// TIA Portal V17 export
// export: Created 2024-08-29T18:23:45.6211091Z, ExportSetting WithDefaults, DisplayName Totally Integrated Automation Portal, DisplayVersion V17 Update 7, DisplayName TIA Portal Openness, DisplayVersion V17 Update 7, DisplayName TIA Portal Version Control Interface, DisplayVersion V17, DisplayName SINAMICS Startdrive Advanced, DisplayVersion V17 SP2, DisplayName SINAMICS Startdrive G110M, G120, G120C, G120D, G120P, G115D, DisplayVersion V17 SP2, DisplayName SINAMICS Startdrive G130, G150, S120, S150, SINAMICS MV, S210, DisplayVersion V17 SP2, DisplayName STEP 7 Professional, DisplayVersion V17 Update 7, DisplayName STEP 7 Safety, DisplayVersion V17 Update 6, DisplayName WinCC Advanced / Unified PC, DisplayVersion V17 Update 7
FUNCTION "sensorStatusArr" : Void   // FC38, LAD
{ S7_Optimized_Access := 'TRUE' }
VERSION : 0.1
// stored: AutoNumber true, IsIECCheckEnabled false, SetENOAutomatically false, UDAEnableTagReadback false
   VAR_INPUT
      manualModeActive : Bool;
      automaticModeActive : Bool;
      sensorRequested : Array[0..31] of Bool;
      sensorActive : Array[0..31] of Bool;
      sensorMask : Array[0..31] of Bool;
   END_VAR
   VAR_OUTPUT
      sensorStatus : Array[0..31] of Byte;
   END_VAR
BEGIN

REGION Network 1: Status 0
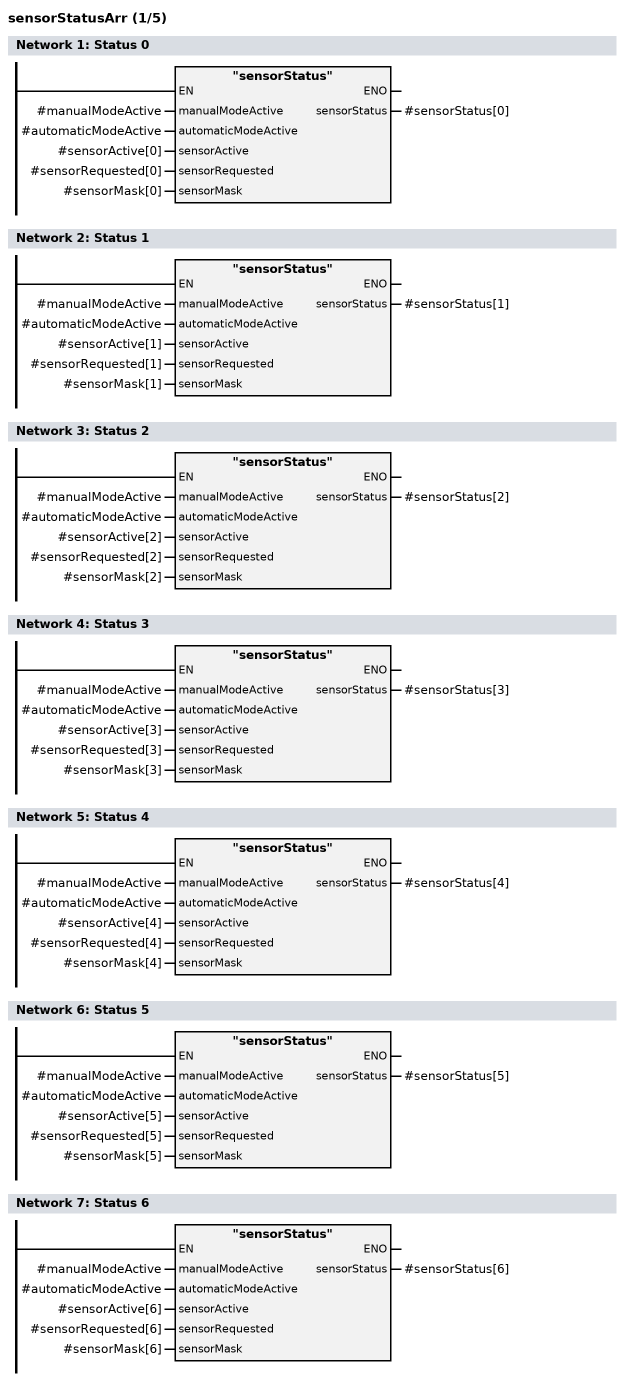
   RUNG wire#powerrail
      "sensorStatus"(manualModeActive := #manualModeActive, automaticModeActive := #automaticModeActive, sensorActive := #sensorActive[0], sensorRequested := #sensorRequested[0], sensorMask := #sensorMask[0], sensorStatus => #sensorStatus[0])
   END_RUNG
   // the same network as SCL:
   "sensorStatus"(manualModeActive := #manualModeActive,
                  automaticModeActive := #automaticModeActive,
                  sensorActive := #sensorActive[0],
                  sensorRequested := #sensorRequested[0],
                  sensorMask := #sensorMask[0],
                  sensorStatus => #sensorStatus[0]);
END_REGION

REGION Network 2: Status 1
   RUNG wire#powerrail
      "sensorStatus"(manualModeActive := #manualModeActive, automaticModeActive := #automaticModeActive, sensorActive := #sensorActive[1], sensorRequested := #sensorRequested[1], sensorMask := #sensorMask[1], sensorStatus => #sensorStatus[1])
   END_RUNG
   // the same network as SCL:
   "sensorStatus"(manualModeActive := #manualModeActive,
                  automaticModeActive := #automaticModeActive,
                  sensorActive := #sensorActive[1],
                  sensorRequested := #sensorRequested[1],
                  sensorMask := #sensorMask[1],
                  sensorStatus => #sensorStatus[1]);
END_REGION

REGION Network 3: Status 2
   RUNG wire#powerrail
      "sensorStatus"(manualModeActive := #manualModeActive, automaticModeActive := #automaticModeActive, sensorActive := #sensorActive[2], sensorRequested := #sensorRequested[2], sensorMask := #sensorMask[2], sensorStatus => #sensorStatus[2])
   END_RUNG
   // the same network as SCL:
   "sensorStatus"(manualModeActive := #manualModeActive,
                  automaticModeActive := #automaticModeActive,
                  sensorActive := #sensorActive[2],
                  sensorRequested := #sensorRequested[2],
                  sensorMask := #sensorMask[2],
                  sensorStatus => #sensorStatus[2]);
END_REGION

REGION Network 4: Status 3
   RUNG wire#powerrail
      "sensorStatus"(manualModeActive := #manualModeActive, automaticModeActive := #automaticModeActive, sensorActive := #sensorActive[3], sensorRequested := #sensorRequested[3], sensorMask := #sensorMask[3], sensorStatus => #sensorStatus[3])
   END_RUNG
   // the same network as SCL:
   "sensorStatus"(manualModeActive := #manualModeActive,
                  automaticModeActive := #automaticModeActive,
                  sensorActive := #sensorActive[3],
                  sensorRequested := #sensorRequested[3],
                  sensorMask := #sensorMask[3],
                  sensorStatus => #sensorStatus[3]);
END_REGION

REGION Network 5: Status 4
   RUNG wire#powerrail
      "sensorStatus"(manualModeActive := #manualModeActive, automaticModeActive := #automaticModeActive, sensorActive := #sensorActive[4], sensorRequested := #sensorRequested[4], sensorMask := #sensorMask[4], sensorStatus => #sensorStatus[4])
   END_RUNG
   // the same network as SCL:
   "sensorStatus"(manualModeActive := #manualModeActive,
                  automaticModeActive := #automaticModeActive,
                  sensorActive := #sensorActive[4],
                  sensorRequested := #sensorRequested[4],
                  sensorMask := #sensorMask[4],
                  sensorStatus => #sensorStatus[4]);
END_REGION

REGION Network 6: Status 5
   RUNG wire#powerrail
      "sensorStatus"(manualModeActive := #manualModeActive, automaticModeActive := #automaticModeActive, sensorActive := #sensorActive[5], sensorRequested := #sensorRequested[5], sensorMask := #sensorMask[5], sensorStatus => #sensorStatus[5])
   END_RUNG
   // the same network as SCL:
   "sensorStatus"(manualModeActive := #manualModeActive,
                  automaticModeActive := #automaticModeActive,
                  sensorActive := #sensorActive[5],
                  sensorRequested := #sensorRequested[5],
                  sensorMask := #sensorMask[5],
                  sensorStatus => #sensorStatus[5]);
END_REGION

REGION Network 7: Status 6
   RUNG wire#powerrail
      "sensorStatus"(manualModeActive := #manualModeActive, automaticModeActive := #automaticModeActive, sensorActive := #sensorActive[6], sensorRequested := #sensorRequested[6], sensorMask := #sensorMask[6], sensorStatus => #sensorStatus[6])
   END_RUNG
   // the same network as SCL:
   "sensorStatus"(manualModeActive := #manualModeActive,
                  automaticModeActive := #automaticModeActive,
                  sensorActive := #sensorActive[6],
                  sensorRequested := #sensorRequested[6],
                  sensorMask := #sensorMask[6],
                  sensorStatus => #sensorStatus[6]);
END_REGION

REGION Network 8: Status 7
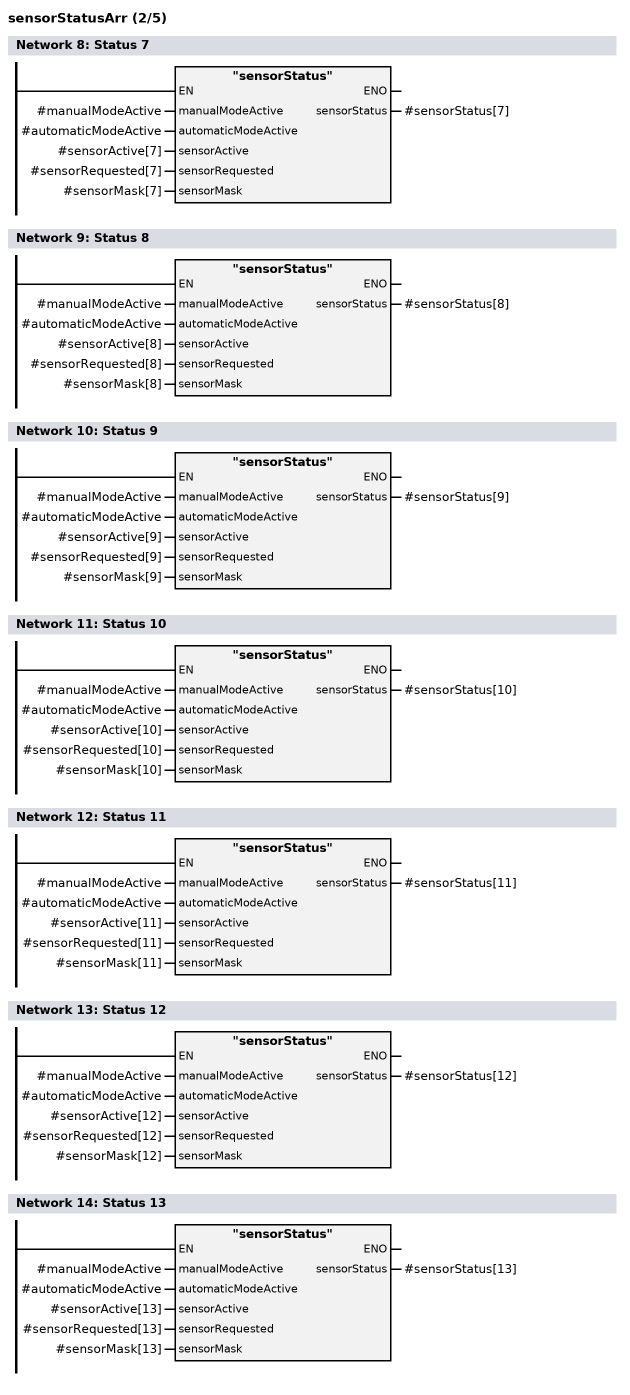
   RUNG wire#powerrail
      "sensorStatus"(manualModeActive := #manualModeActive, automaticModeActive := #automaticModeActive, sensorActive := #sensorActive[7], sensorRequested := #sensorRequested[7], sensorMask := #sensorMask[7], sensorStatus => #sensorStatus[7])
   END_RUNG
   // the same network as SCL:
   "sensorStatus"(manualModeActive := #manualModeActive,
                  automaticModeActive := #automaticModeActive,
                  sensorActive := #sensorActive[7],
                  sensorRequested := #sensorRequested[7],
                  sensorMask := #sensorMask[7],
                  sensorStatus => #sensorStatus[7]);
END_REGION

REGION Network 9: Status 8
   RUNG wire#powerrail
      "sensorStatus"(manualModeActive := #manualModeActive, automaticModeActive := #automaticModeActive, sensorActive := #sensorActive[8], sensorRequested := #sensorRequested[8], sensorMask := #sensorMask[8], sensorStatus => #sensorStatus[8])
   END_RUNG
   // the same network as SCL:
   "sensorStatus"(manualModeActive := #manualModeActive,
                  automaticModeActive := #automaticModeActive,
                  sensorActive := #sensorActive[8],
                  sensorRequested := #sensorRequested[8],
                  sensorMask := #sensorMask[8],
                  sensorStatus => #sensorStatus[8]);
END_REGION

REGION Network 10: Status 9
   RUNG wire#powerrail
      "sensorStatus"(manualModeActive := #manualModeActive, automaticModeActive := #automaticModeActive, sensorActive := #sensorActive[9], sensorRequested := #sensorRequested[9], sensorMask := #sensorMask[9], sensorStatus => #sensorStatus[9])
   END_RUNG
   // the same network as SCL:
   "sensorStatus"(manualModeActive := #manualModeActive,
                  automaticModeActive := #automaticModeActive,
                  sensorActive := #sensorActive[9],
                  sensorRequested := #sensorRequested[9],
                  sensorMask := #sensorMask[9],
                  sensorStatus => #sensorStatus[9]);
END_REGION

REGION Network 11: Status 10
   RUNG wire#powerrail
      "sensorStatus"(manualModeActive := #manualModeActive, automaticModeActive := #automaticModeActive, sensorActive := #sensorActive[10], sensorRequested := #sensorRequested[10], sensorMask := #sensorMask[10], sensorStatus => #sensorStatus[10])
   END_RUNG
   // the same network as SCL:
   "sensorStatus"(manualModeActive := #manualModeActive,
                  automaticModeActive := #automaticModeActive,
                  sensorActive := #sensorActive[10],
                  sensorRequested := #sensorRequested[10],
                  sensorMask := #sensorMask[10],
                  sensorStatus => #sensorStatus[10]);
END_REGION

REGION Network 12: Status 11
   RUNG wire#powerrail
      "sensorStatus"(manualModeActive := #manualModeActive, automaticModeActive := #automaticModeActive, sensorActive := #sensorActive[11], sensorRequested := #sensorRequested[11], sensorMask := #sensorMask[11], sensorStatus => #sensorStatus[11])
   END_RUNG
   // the same network as SCL:
   "sensorStatus"(manualModeActive := #manualModeActive,
                  automaticModeActive := #automaticModeActive,
                  sensorActive := #sensorActive[11],
                  sensorRequested := #sensorRequested[11],
                  sensorMask := #sensorMask[11],
                  sensorStatus => #sensorStatus[11]);
END_REGION

REGION Network 13: Status 12
   RUNG wire#powerrail
      "sensorStatus"(manualModeActive := #manualModeActive, automaticModeActive := #automaticModeActive, sensorActive := #sensorActive[12], sensorRequested := #sensorRequested[12], sensorMask := #sensorMask[12], sensorStatus => #sensorStatus[12])
   END_RUNG
   // the same network as SCL:
   "sensorStatus"(manualModeActive := #manualModeActive,
                  automaticModeActive := #automaticModeActive,
                  sensorActive := #sensorActive[12],
                  sensorRequested := #sensorRequested[12],
                  sensorMask := #sensorMask[12],
                  sensorStatus => #sensorStatus[12]);
END_REGION

REGION Network 14: Status 13
   RUNG wire#powerrail
      "sensorStatus"(manualModeActive := #manualModeActive, automaticModeActive := #automaticModeActive, sensorActive := #sensorActive[13], sensorRequested := #sensorRequested[13], sensorMask := #sensorMask[13], sensorStatus => #sensorStatus[13])
   END_RUNG
   // the same network as SCL:
   "sensorStatus"(manualModeActive := #manualModeActive,
                  automaticModeActive := #automaticModeActive,
                  sensorActive := #sensorActive[13],
                  sensorRequested := #sensorRequested[13],
                  sensorMask := #sensorMask[13],
                  sensorStatus => #sensorStatus[13]);
END_REGION

REGION Network 15: Status 14
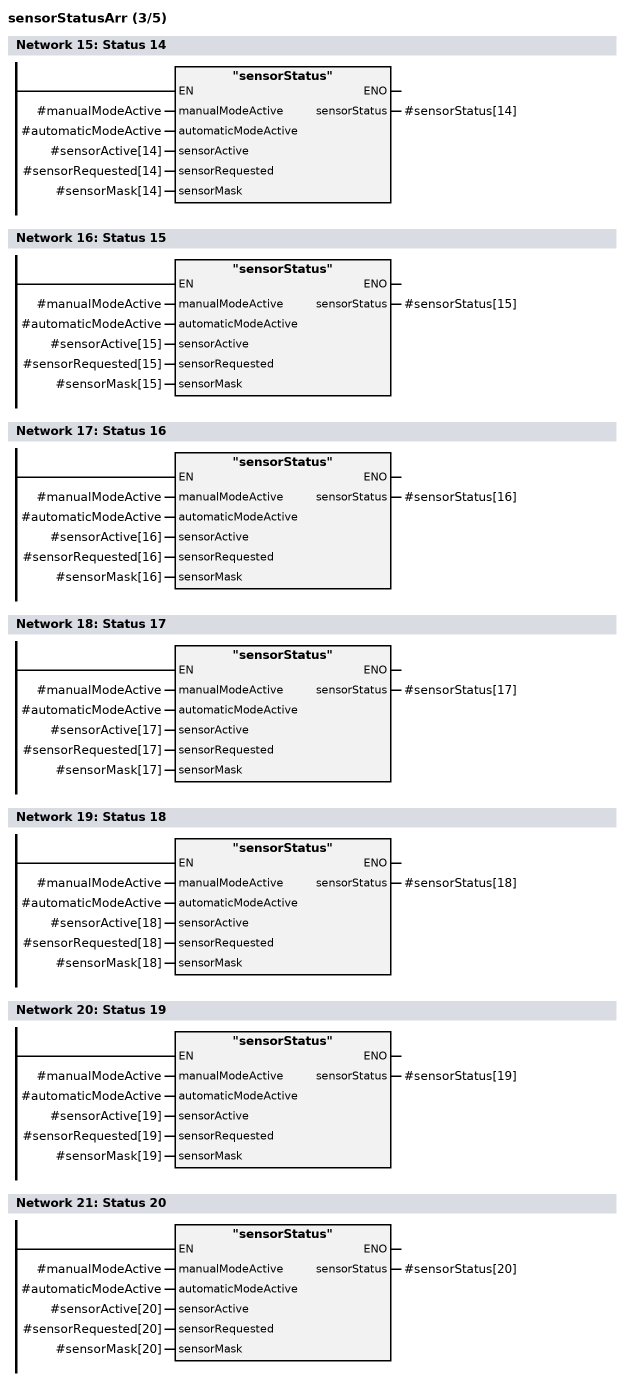
   RUNG wire#powerrail
      "sensorStatus"(manualModeActive := #manualModeActive, automaticModeActive := #automaticModeActive, sensorActive := #sensorActive[14], sensorRequested := #sensorRequested[14], sensorMask := #sensorMask[14], sensorStatus => #sensorStatus[14])
   END_RUNG
   // the same network as SCL:
   "sensorStatus"(manualModeActive := #manualModeActive,
                  automaticModeActive := #automaticModeActive,
                  sensorActive := #sensorActive[14],
                  sensorRequested := #sensorRequested[14],
                  sensorMask := #sensorMask[14],
                  sensorStatus => #sensorStatus[14]);
END_REGION

REGION Network 16: Status 15
   RUNG wire#powerrail
      "sensorStatus"(manualModeActive := #manualModeActive, automaticModeActive := #automaticModeActive, sensorActive := #sensorActive[15], sensorRequested := #sensorRequested[15], sensorMask := #sensorMask[15], sensorStatus => #sensorStatus[15])
   END_RUNG
   // the same network as SCL:
   "sensorStatus"(manualModeActive := #manualModeActive,
                  automaticModeActive := #automaticModeActive,
                  sensorActive := #sensorActive[15],
                  sensorRequested := #sensorRequested[15],
                  sensorMask := #sensorMask[15],
                  sensorStatus => #sensorStatus[15]);
END_REGION

REGION Network 17: Status 16
   RUNG wire#powerrail
      "sensorStatus"(manualModeActive := #manualModeActive, automaticModeActive := #automaticModeActive, sensorActive := #sensorActive[16], sensorRequested := #sensorRequested[16], sensorMask := #sensorMask[16], sensorStatus => #sensorStatus[16])
   END_RUNG
   // the same network as SCL:
   "sensorStatus"(manualModeActive := #manualModeActive,
                  automaticModeActive := #automaticModeActive,
                  sensorActive := #sensorActive[16],
                  sensorRequested := #sensorRequested[16],
                  sensorMask := #sensorMask[16],
                  sensorStatus => #sensorStatus[16]);
END_REGION

REGION Network 18: Status 17
   RUNG wire#powerrail
      "sensorStatus"(manualModeActive := #manualModeActive, automaticModeActive := #automaticModeActive, sensorActive := #sensorActive[17], sensorRequested := #sensorRequested[17], sensorMask := #sensorMask[17], sensorStatus => #sensorStatus[17])
   END_RUNG
   // the same network as SCL:
   "sensorStatus"(manualModeActive := #manualModeActive,
                  automaticModeActive := #automaticModeActive,
                  sensorActive := #sensorActive[17],
                  sensorRequested := #sensorRequested[17],
                  sensorMask := #sensorMask[17],
                  sensorStatus => #sensorStatus[17]);
END_REGION

REGION Network 19: Status 18
   RUNG wire#powerrail
      "sensorStatus"(manualModeActive := #manualModeActive, automaticModeActive := #automaticModeActive, sensorActive := #sensorActive[18], sensorRequested := #sensorRequested[18], sensorMask := #sensorMask[18], sensorStatus => #sensorStatus[18])
   END_RUNG
   // the same network as SCL:
   "sensorStatus"(manualModeActive := #manualModeActive,
                  automaticModeActive := #automaticModeActive,
                  sensorActive := #sensorActive[18],
                  sensorRequested := #sensorRequested[18],
                  sensorMask := #sensorMask[18],
                  sensorStatus => #sensorStatus[18]);
END_REGION

REGION Network 20: Status 19
   RUNG wire#powerrail
      "sensorStatus"(manualModeActive := #manualModeActive, automaticModeActive := #automaticModeActive, sensorActive := #sensorActive[19], sensorRequested := #sensorRequested[19], sensorMask := #sensorMask[19], sensorStatus => #sensorStatus[19])
   END_RUNG
   // the same network as SCL:
   "sensorStatus"(manualModeActive := #manualModeActive,
                  automaticModeActive := #automaticModeActive,
                  sensorActive := #sensorActive[19],
                  sensorRequested := #sensorRequested[19],
                  sensorMask := #sensorMask[19],
                  sensorStatus => #sensorStatus[19]);
END_REGION

REGION Network 21: Status 20
   RUNG wire#powerrail
      "sensorStatus"(manualModeActive := #manualModeActive, automaticModeActive := #automaticModeActive, sensorActive := #sensorActive[20], sensorRequested := #sensorRequested[20], sensorMask := #sensorMask[20], sensorStatus => #sensorStatus[20])
   END_RUNG
   // the same network as SCL:
   "sensorStatus"(manualModeActive := #manualModeActive,
                  automaticModeActive := #automaticModeActive,
                  sensorActive := #sensorActive[20],
                  sensorRequested := #sensorRequested[20],
                  sensorMask := #sensorMask[20],
                  sensorStatus => #sensorStatus[20]);
END_REGION

REGION Network 22: Status 21
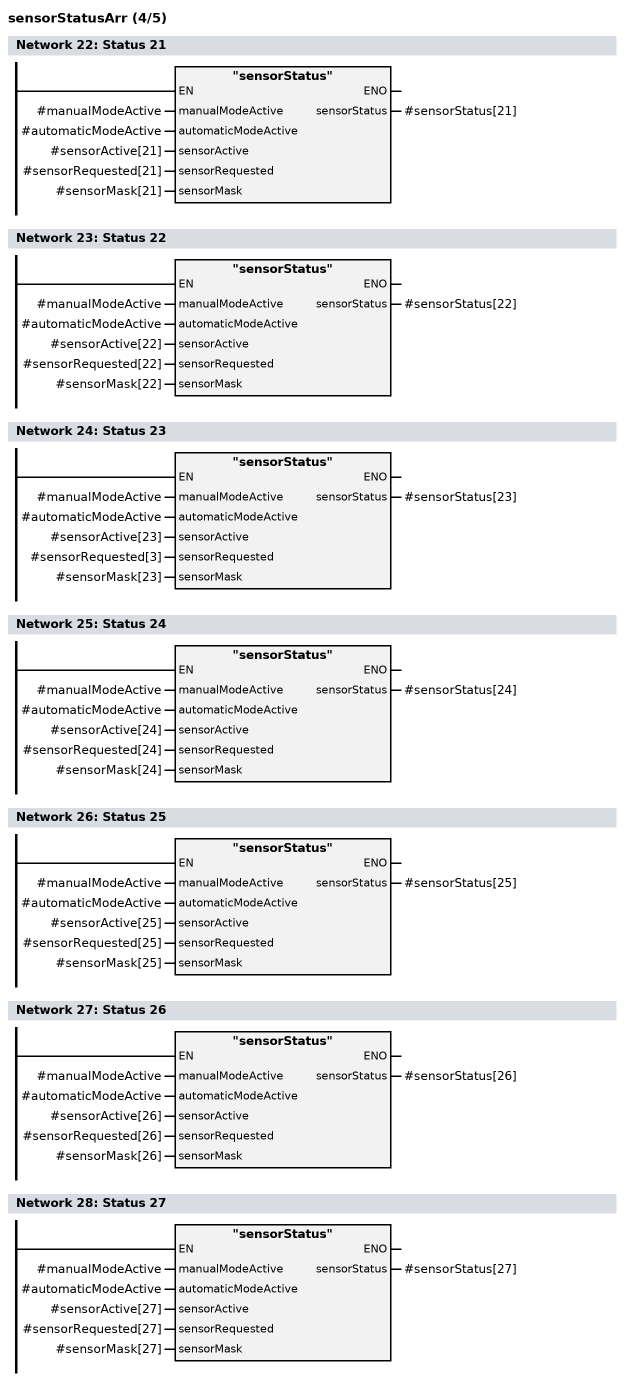
   RUNG wire#powerrail
      "sensorStatus"(manualModeActive := #manualModeActive, automaticModeActive := #automaticModeActive, sensorActive := #sensorActive[21], sensorRequested := #sensorRequested[21], sensorMask := #sensorMask[21], sensorStatus => #sensorStatus[21])
   END_RUNG
   // the same network as SCL:
   "sensorStatus"(manualModeActive := #manualModeActive,
                  automaticModeActive := #automaticModeActive,
                  sensorActive := #sensorActive[21],
                  sensorRequested := #sensorRequested[21],
                  sensorMask := #sensorMask[21],
                  sensorStatus => #sensorStatus[21]);
END_REGION

REGION Network 23: Status 22
   RUNG wire#powerrail
      "sensorStatus"(manualModeActive := #manualModeActive, automaticModeActive := #automaticModeActive, sensorActive := #sensorActive[22], sensorRequested := #sensorRequested[22], sensorMask := #sensorMask[22], sensorStatus => #sensorStatus[22])
   END_RUNG
   // the same network as SCL:
   "sensorStatus"(manualModeActive := #manualModeActive,
                  automaticModeActive := #automaticModeActive,
                  sensorActive := #sensorActive[22],
                  sensorRequested := #sensorRequested[22],
                  sensorMask := #sensorMask[22],
                  sensorStatus => #sensorStatus[22]);
END_REGION

REGION Network 24: Status 23
   RUNG wire#powerrail
      "sensorStatus"(manualModeActive := #manualModeActive, automaticModeActive := #automaticModeActive, sensorActive := #sensorActive[23], sensorRequested := #sensorRequested[3], sensorMask := #sensorMask[23], sensorStatus => #sensorStatus[23])
   END_RUNG
   // the same network as SCL:
   "sensorStatus"(manualModeActive := #manualModeActive,
                  automaticModeActive := #automaticModeActive,
                  sensorActive := #sensorActive[23],
                  sensorRequested := #sensorRequested[3],
                  sensorMask := #sensorMask[23],
                  sensorStatus => #sensorStatus[23]);
END_REGION

REGION Network 25: Status 24
   RUNG wire#powerrail
      "sensorStatus"(manualModeActive := #manualModeActive, automaticModeActive := #automaticModeActive, sensorActive := #sensorActive[24], sensorRequested := #sensorRequested[24], sensorMask := #sensorMask[24], sensorStatus => #sensorStatus[24])
   END_RUNG
   // the same network as SCL:
   "sensorStatus"(manualModeActive := #manualModeActive,
                  automaticModeActive := #automaticModeActive,
                  sensorActive := #sensorActive[24],
                  sensorRequested := #sensorRequested[24],
                  sensorMask := #sensorMask[24],
                  sensorStatus => #sensorStatus[24]);
END_REGION

REGION Network 26: Status 25
   RUNG wire#powerrail
      "sensorStatus"(manualModeActive := #manualModeActive, automaticModeActive := #automaticModeActive, sensorActive := #sensorActive[25], sensorRequested := #sensorRequested[25], sensorMask := #sensorMask[25], sensorStatus => #sensorStatus[25])
   END_RUNG
   // the same network as SCL:
   "sensorStatus"(manualModeActive := #manualModeActive,
                  automaticModeActive := #automaticModeActive,
                  sensorActive := #sensorActive[25],
                  sensorRequested := #sensorRequested[25],
                  sensorMask := #sensorMask[25],
                  sensorStatus => #sensorStatus[25]);
END_REGION

REGION Network 27: Status 26
   RUNG wire#powerrail
      "sensorStatus"(manualModeActive := #manualModeActive, automaticModeActive := #automaticModeActive, sensorActive := #sensorActive[26], sensorRequested := #sensorRequested[26], sensorMask := #sensorMask[26], sensorStatus => #sensorStatus[26])
   END_RUNG
   // the same network as SCL:
   "sensorStatus"(manualModeActive := #manualModeActive,
                  automaticModeActive := #automaticModeActive,
                  sensorActive := #sensorActive[26],
                  sensorRequested := #sensorRequested[26],
                  sensorMask := #sensorMask[26],
                  sensorStatus => #sensorStatus[26]);
END_REGION

REGION Network 28: Status 27
   RUNG wire#powerrail
      "sensorStatus"(manualModeActive := #manualModeActive, automaticModeActive := #automaticModeActive, sensorActive := #sensorActive[27], sensorRequested := #sensorRequested[27], sensorMask := #sensorMask[27], sensorStatus => #sensorStatus[27])
   END_RUNG
   // the same network as SCL:
   "sensorStatus"(manualModeActive := #manualModeActive,
                  automaticModeActive := #automaticModeActive,
                  sensorActive := #sensorActive[27],
                  sensorRequested := #sensorRequested[27],
                  sensorMask := #sensorMask[27],
                  sensorStatus => #sensorStatus[27]);
END_REGION

REGION Network 29: Status 28
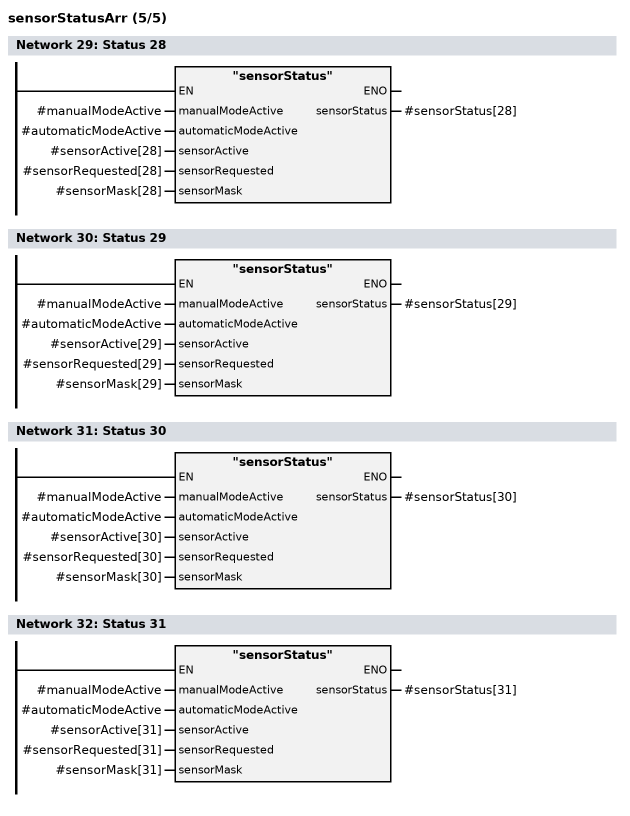
   RUNG wire#powerrail
      "sensorStatus"(manualModeActive := #manualModeActive, automaticModeActive := #automaticModeActive, sensorActive := #sensorActive[28], sensorRequested := #sensorRequested[28], sensorMask := #sensorMask[28], sensorStatus => #sensorStatus[28])
   END_RUNG
   // the same network as SCL:
   "sensorStatus"(manualModeActive := #manualModeActive,
                  automaticModeActive := #automaticModeActive,
                  sensorActive := #sensorActive[28],
                  sensorRequested := #sensorRequested[28],
                  sensorMask := #sensorMask[28],
                  sensorStatus => #sensorStatus[28]);
END_REGION

REGION Network 30: Status 29
   RUNG wire#powerrail
      "sensorStatus"(manualModeActive := #manualModeActive, automaticModeActive := #automaticModeActive, sensorActive := #sensorActive[29], sensorRequested := #sensorRequested[29], sensorMask := #sensorMask[29], sensorStatus => #sensorStatus[29])
   END_RUNG
   // the same network as SCL:
   "sensorStatus"(manualModeActive := #manualModeActive,
                  automaticModeActive := #automaticModeActive,
                  sensorActive := #sensorActive[29],
                  sensorRequested := #sensorRequested[29],
                  sensorMask := #sensorMask[29],
                  sensorStatus => #sensorStatus[29]);
END_REGION

REGION Network 31: Status 30
   RUNG wire#powerrail
      "sensorStatus"(manualModeActive := #manualModeActive, automaticModeActive := #automaticModeActive, sensorActive := #sensorActive[30], sensorRequested := #sensorRequested[30], sensorMask := #sensorMask[30], sensorStatus => #sensorStatus[30])
   END_RUNG
   // the same network as SCL:
   "sensorStatus"(manualModeActive := #manualModeActive,
                  automaticModeActive := #automaticModeActive,
                  sensorActive := #sensorActive[30],
                  sensorRequested := #sensorRequested[30],
                  sensorMask := #sensorMask[30],
                  sensorStatus => #sensorStatus[30]);
END_REGION

REGION Network 32: Status 31
   RUNG wire#powerrail
      "sensorStatus"(manualModeActive := #manualModeActive, automaticModeActive := #automaticModeActive, sensorActive := #sensorActive[31], sensorRequested := #sensorRequested[31], sensorMask := #sensorMask[31], sensorStatus => #sensorStatus[31])
   END_RUNG
   // the same network as SCL:
   "sensorStatus"(manualModeActive := #manualModeActive,
                  automaticModeActive := #automaticModeActive,
                  sensorActive := #sensorActive[31],
                  sensorRequested := #sensorRequested[31],
                  sensorMask := #sensorMask[31],
                  sensorStatus => #sensorStatus[31]);
END_REGION
END_FUNCTION
